# EPICS autosave request: ADApp/Db/NDPva_settings.req
# Nothing extra needed beyond NDPluginBase_settings.req for now
file "NDPluginBase_settings.req", P=$(P), R=$(R)
